GLOBALCONSTANTS DefaultPool (* Global constants *)
  PACKAGE Uebungen::const::UT::Scroll;
  VAR_GLOBAL CONSTANT
    ISO_DESIGNATOR_WIDTH : UINT := 80;
    ISO_DESIGNATOR_HEIGHT : UINT := 80;
    ISO_MASK_SIZE : UINT := 480;
    ISO_VERSION_LABEL : STRING;
    MASK_WIDTH : UINT := 480;
    MASK_HEIGHT : UINT := 480;
    WorkingSet : UINT := 0;
    MainMask : UINT := 1000;
    DataMask_invisible : UINT := 1001;
    Container_Scrollbar_Parent : UINT := 3000;
    Container_3001 : UINT := 3001;
    Container_3002 : UINT := 3002;
    Container_3003 : UINT := 3003;
    Container_Dialog_Speichern : UINT := 3004;
    Container_page_header : UINT := 3005;
    Containerr_Scrolling_Parent : UINT := 3006;
    Container_Row_01 : UINT := 3007;
    Container_3008 : UINT := 3008;
    Container_Row_02 : UINT := 3009;
    Container_Scrollbar_Content : UINT := 3010;
    Container_3020 : UINT := 3020;
    Container_3021 : UINT := 3021;
    Container_3022 : UINT := 3022;
    Container_3023 : UINT := 3023;
    Container_Scrolling_Content : UINT := 3031;
    Container_Row_03 : UINT := 3032;
    Container_Row_04 : UINT := 3033;
    Container_Row_05 : UINT := 3034;
    Container_Row_06 : UINT := 3035;
    Container_Row_07 : UINT := 3036;
    Container_Row_08 : UINT := 3037;
    Container_Row_09 : UINT := 3038;
    Container_Row_10 : UINT := 3039;
    Container_Row_11 : UINT := 3040;
    Container_Row_12 : UINT := 3041;
    Container_Row_13 : UINT := 3042;
    Container_Row_14 : UINT := 3043;
    Container_Row_15 : UINT := 3044;
    Container_Row_16 : UINT := 3045;
    Container_Row_17 : UINT := 3046;
    Container_Row_18 : UINT := 3047;
    Container_Row_19 : UINT := 3048;
    Container_Row_20 : UINT := 3049;
    Container_Row_03_Sub : UINT := 3050;
    Container_Row_04_Sub : UINT := 3051;
    Container_Row_05_Sub : UINT := 3052;
    Container_Row_06_Sub : UINT := 3053;
    Container_Row_07_Sub : UINT := 3054;
    Container_Row_08_Sub : UINT := 3055;
    Container_Row_09_Sub : UINT := 3056;
    Container_Row_10_Sub : UINT := 3057;
    Container_Row_11_Sub : UINT := 3058;
    Container_Row_12_Sub : UINT := 3059;
    Container_Row_13_Sub : UINT := 3060;
    Container_Row_14_Sub : UINT := 3061;
    Container_Row_15_Sub : UINT := 3062;
    Container_Row_16_Sub : UINT := 3063;
    Container_Row_17_Sub : UINT := 3064;
    Container_Row_18_Sub : UINT := 3065;
    Container_Row_19_Sub : UINT := 3066;
    Container_Row_20_Sub : UINT := 3067;
    MainSoftKeyMask : UINT := 4000;
    SoftKey_Back : UINT := 5000;
    SoftKey_Lock : UINT := 5001;
    SoftKey_UP_UP : UINT := 5002;
    SoftKey_UP : UINT := 5003;
    SoftKey_DOWN : UINT := 5004;
    SoftKey_DOWN_DOWN : UINT := 5005;
    Button_6000 : UINT := 6000;
    Button_6001 : UINT := 6001;
    Button_6009 : UINT := 6009;
    Button_6010 : UINT := 6010;
    OutputString_11000 : UINT := 11000;
    OutputString_11001 : UINT := 11001;
    OutputString_Label_01 : UINT := 11002;
    OutputString_11003 : UINT := 11003;
    OutputString_11004 : UINT := 11004;
    OutputString_11005 : UINT := 11005;
    OutputString_11006 : UINT := 11006;
    OutputString_Label_01_long : UINT := 11009;
    OutputString_11016 : UINT := 11016;
    OutputString_11023 : UINT := 11023;
    OutputString_Werte_speichern : UINT := 11030;
    OutputString_Row_03_Label : UINT := 11031;
    OutputString_Row_04_Label : UINT := 11032;
    OutputString_Row_05_Label : UINT := 11033;
    OutputString_Row_06_Label : UINT := 11034;
    OutputString_Row_07_Label : UINT := 11035;
    OutputString_Row_08_Label : UINT := 11036;
    OutputString_Row_09_Label : UINT := 11037;
    OutputString_Row_10_Label : UINT := 11038;
    OutputString_Row_11_Label : UINT := 11039;
    OutputString_Row_12_Label : UINT := 11040;
    OutputString_Row_13_Label : UINT := 11041;
    OutputString_Row_14_Label : UINT := 11042;
    OutputString_Row_15_Label : UINT := 11043;
    OutputString_Row_16_Label : UINT := 11044;
    OutputString_Row_17_Label : UINT := 11045;
    OutputString_Row_18_Label : UINT := 11046;
    OutputString_Row_19_Label : UINT := 11047;
    OutputString_Row_20_Label : UINT := 11048;
    OutputString_Row_03_Name : UINT := 11049;
    OutputString_Row_04_Name : UINT := 11050;
    OutputString_Row_05_Name : UINT := 11051;
    OutputString_Row_06_Name : UINT := 11052;
    OutputString_Row_07_Name : UINT := 11053;
    OutputString_Row_08_Name : UINT := 11054;
    OutputString_Row_09_Name : UINT := 11055;
    OutputString_Row_10_Name : UINT := 11056;
    OutputString_Row_11_Name : UINT := 11057;
    OutputString_Row_12_Name : UINT := 11058;
    OutputString_Row_13_Name : UINT := 11059;
    OutputString_Row_14_Name : UINT := 11060;
    OutputString_Row_15_Name : UINT := 11061;
    OutputString_Row_16_Name : UINT := 11062;
    OutputString_Row_17_Name : UINT := 11063;
    OutputString_Row_18_Name : UINT := 11064;
    OutputString_Row_19_Name : UINT := 11065;
    OutputString_Row_20_Name : UINT := 11066;
    OutputString_Row_03_Unit : UINT := 11067;
    OutputString_Row_04_Unit : UINT := 11068;
    OutputString_Row_05_Unit : UINT := 11069;
    OutputString_Row_06_Unit : UINT := 11070;
    OutputString_Row_07_Unit : UINT := 11071;
    OutputString_Row_08_Unit : UINT := 11072;
    OutputString_Row_09_Unit : UINT := 11073;
    OutputString_Row_10_Unit : UINT := 11074;
    OutputString_Row_11_Unit : UINT := 11075;
    OutputString_Row_12_Unit : UINT := 11076;
    OutputString_Row_13_Unit : UINT := 11077;
    OutputString_Row_14_Unit : UINT := 11078;
    OutputString_Row_15_Unit : UINT := 11079;
    OutputString_Row_16_Unit : UINT := 11080;
    OutputString_Row_17_Unit : UINT := 11081;
    OutputString_Row_18_Unit : UINT := 11082;
    OutputString_Row_19_Unit : UINT := 11083;
    OutputString_Row_20_Unit : UINT := 11084;
    OutputString_Row_03_SubText : UINT := 11085;
    OutputString_Row_04_SubText : UINT := 11086;
    OutputString_Row_05_SubText : UINT := 11087;
    OutputString_Row_06_SubText : UINT := 11088;
    OutputString_Row_07_SubText : UINT := 11089;
    OutputString_Row_08_SubText : UINT := 11090;
    OutputString_Row_09_SubText : UINT := 11091;
    OutputString_Row_10_SubText : UINT := 11092;
    OutputString_Row_11_SubText : UINT := 11093;
    OutputString_Row_12_SubText : UINT := 11094;
    OutputString_Row_13_SubText : UINT := 11095;
    OutputString_Row_14_SubText : UINT := 11096;
    OutputString_Row_15_SubText : UINT := 11097;
    OutputString_Row_16_SubText : UINT := 11098;
    OutputString_Row_17_SubText : UINT := 11099;
    OutputString_Row_18_SubText : UINT := 11100;
    OutputString_Row_19_SubText : UINT := 11101;
    OutputString_Row_20_SubText : UINT := 11102;
    OutputNumber_12000 : UINT := 12000;
    OutputNumber_old_value : UINT := 12001;
    OutputNumber_12002 : UINT := 12002;
    OutputNumber_12003 : UINT := 12003;
    OutputNumber_new_value : UINT := 12008;
    OutputNumber_Row_03_Value : UINT := 12009;
    OutputNumber_Row_04_Value : UINT := 12010;
    OutputNumber_Row_05_Value : UINT := 12011;
    OutputNumber_Row_06_Value : UINT := 12012;
    OutputNumber_Row_07_Value : UINT := 12013;
    OutputNumber_Row_08_Value : UINT := 12014;
    OutputNumber_Row_09_Value : UINT := 12015;
    OutputNumber_Row_10_Value : UINT := 12016;
    OutputNumber_Row_11_Value : UINT := 12017;
    OutputNumber_Row_12_Value : UINT := 12018;
    OutputNumber_Row_13_Value : UINT := 12019;
    OutputNumber_Row_14_Value : UINT := 12020;
    OutputNumber_Row_15_Value : UINT := 12021;
    OutputNumber_Row_16_Value : UINT := 12022;
    OutputNumber_Row_17_Value : UINT := 12023;
    OutputNumber_Row_18_Value : UINT := 12024;
    OutputNumber_Row_19_Value : UINT := 12025;
    OutputNumber_Row_20_Value : UINT := 12026;
    OutputNumber_Row_03_SubValue : UINT := 12027;
    OutputNumber_Row_04_SubValue : UINT := 12028;
    OutputNumber_Row_05_SubValue : UINT := 12029;
    OutputNumber_Row_06_SubValue : UINT := 12030;
    OutputNumber_Row_07_SubValue : UINT := 12031;
    OutputNumber_Row_08_SubValue : UINT := 12032;
    OutputNumber_Row_09_SubValue : UINT := 12033;
    OutputNumber_Row_10_SubValue : UINT := 12034;
    OutputNumber_Row_11_SubValue : UINT := 12035;
    OutputNumber_Row_12_SubValue : UINT := 12036;
    OutputNumber_Row_13_SubValue : UINT := 12037;
    OutputNumber_Row_14_SubValue : UINT := 12038;
    OutputNumber_Row_15_SubValue : UINT := 12039;
    OutputNumber_Row_16_SubValue : UINT := 12040;
    OutputNumber_Row_17_SubValue : UINT := 12041;
    OutputNumber_Row_18_SubValue : UINT := 12042;
    OutputNumber_Row_19_SubValue : UINT := 12043;
    OutputNumber_Row_20_SubValue : UINT := 12044;
    Line : UINT := 13000;
    Rectangle_Scrollbar : UINT := 14000;
    Rectangle_Scroll_Indicator : UINT := 14001;
    Rectangle_14002 : UINT := 14002;
    Rectangle_14003 : UINT := 14003;
    Rectangle_14004 : UINT := 14004;
    Rectangle_14005 : UINT := 14005;
    Rectangle_14006 : UINT := 14006;
    Rectangle_14013 : UINT := 14013;
    Rectangle_grey : UINT := 14014;
    Rectangle_14015 : UINT := 14015;
    Rectangle_14028 : UINT := 14028;
    Rectangle_14029 : UINT := 14029;
    Rectangle_14107 : UINT := 14107;
    Image_20000 : UINT := 20000;
    Image_20001 : UINT := 20001;
    Image_20002 : UINT := 20002;
    Image_20003 : UINT := 20003;
    Image_20086 : UINT := 20004;
    Image_55027_20005 : UINT := 20005;
    Image_55027_20006 : UINT := 20006;
    Image_55028_20007 : UINT := 20007;
    Image_55028_20008 : UINT := 20008;
    Image_55028_20009 : UINT := 20009;
    Image_55027_20010 : UINT := 20010;
    Image_20343 : UINT := 20011;
    Image_20329 : UINT := 20329;
    StringVariable_22000 : UINT := 22000;
    StringVariable_22001 : UINT := 22001;
    StringVariable_22008 : UINT := 22008;
    StringVariable_22009 : UINT := 22009;
    StringVariable_22010 : UINT := 22010;
    StringVariable_22011 : UINT := 22011;
    StringVariable_22012 : UINT := 22012;
    StringVariable_22013 : UINT := 22013;
    StringVariable_22014 : UINT := 22014;
    StringVariable_22015 : UINT := 22015;
    StringVariable_22016 : UINT := 22016;
    StringVariable_22017 : UINT := 22017;
    StringVariable_22018 : UINT := 22018;
    StringVariable_22019 : UINT := 22019;
    StringVariable_22020 : UINT := 22020;
    StringVariable_22021 : UINT := 22021;
    StringVariable_22022 : UINT := 22022;
    StringVariable_22023 : UINT := 22023;
    StringVariable_22024 : UINT := 22024;
    StringVariable_22025 : UINT := 22025;
    StringVariable_22026 : UINT := 22026;
    FontAttributes_8x12 : UINT := 23000;
    FontAttributes_23001 : UINT := 23001;
    FontAttributes_23002 : UINT := 23002;
    FontAttributes_23003 : UINT := 23003;
    FontAttributes_23004 : UINT := 23004;
    FontAttributes_23005 : UINT := 23005;
    LineAttributes_white : UINT := 24000;
    LineAttributes_24001 : UINT := 24001;
    LineAttributes_24002 : UINT := 24002;
    LineAttributes_24003 : UINT := 24003;
    LineAttributes_24004 : UINT := 24004;
    LineAttributes_24005 : UINT := 24005;
    LineAttributes_24006 : UINT := 24006;
    LineAttributes_grey : UINT := 24007;
    LineAttributes_24018 : UINT := 24018;
    LineAttributes_24019 : UINT := 24019;
    FillAttributes_25000 : UINT := 25000;
    FillAttributes_25001 : UINT := 25001;
    FillAttributes_25002 : UINT := 25002;
    FillAttributes_25003 : UINT := 25003;
    FillAttributes_grey : UINT := 25004;
    FillAttributes_25005 : UINT := 25005;
    FillAttributes_25006 : UINT := 25006;
    FillAttributes_white : UINT := 25007;
    FillAttributes_25020 : UINT := 25020;
    ObjectPointer_Container_Dialog_Speichern : UINT := 27000;
    ObjectPointer_27001 : UINT := 27001;
    ObjectPointer_27002 : UINT := 27002;
    ObjectPointer_27003 : UINT := 27003;
    ObjectPointer_27004 : UINT := 27004;
    ObjectPointer_27005 : UINT := 27005;
    ObjectPointer_Row_03_Status : UINT := 27006;
    ObjectPointer_Row_04_Status : UINT := 27007;
    ObjectPointer_Row_05_Status : UINT := 27008;
    ObjectPointer_Row_06_Status : UINT := 27009;
    ObjectPointer_Row_07_Status : UINT := 27010;
    ObjectPointer_Row_08_Status : UINT := 27011;
    ObjectPointer_Row_09_Status : UINT := 27012;
    ObjectPointer_Row_10_Status : UINT := 27013;
    ObjectPointer_Row_11_Status : UINT := 27014;
    ObjectPointer_Row_12_Status : UINT := 27015;
    ObjectPointer_Row_13_Status : UINT := 27016;
    ObjectPointer_Row_14_Status : UINT := 27017;
    ObjectPointer_Row_15_Status : UINT := 27018;
    ObjectPointer_Row_16_Status : UINT := 27019;
    ObjectPointer_Row_17_Status : UINT := 27020;
    ObjectPointer_Row_18_Status : UINT := 27021;
    ObjectPointer_Row_19_Status : UINT := 27022;
    ObjectPointer_Row_20_Status : UINT := 27023;
    ObjectPointer_SoftKey_Back : UINT := 27024;
    ObjectPointer_27025 : UINT := 27025;
    ObjectPointer_27026 : UINT := 27026;
    ObjectPointer_27027 : UINT := 27027;
    ObjectPointer_27028 : UINT := 27028;
    ObjectPointer_27029 : UINT := 27029;
  END_VAR
END_GLOBALCONSTANTS
